ABB RobotStudio station: Lab3.rsstn

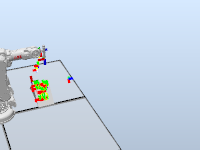
Station Lab1 (saved by RobotStudio 22.1.9826.0)
Controller IRB140_6_81
  mechanical unit ROB_1: IRB140_6_81_C_03, 6 joints, base frame (0, 0, 0) mm
Layout (positions relative to the parent item):
  - IRB140_6_81_C_03 [mechanism, from Robots\IRB140_6_81_C_G_03.rslib] at (0, 0, 0) mm; joint values [0.1206, 0.0069, 0.5145, 0.2099, -0.5334, 0.5073] (rad or m)
  - TableroBorrable [part, from Libraries\TableroBorrable.rslib] at (618.49, 141.25, 150.15) mm
  - Portamarcador [mechanism, from Libraries\Portamarcador.rslib] at (515, 0, 712) mm, rotated rx 0 ry 90 rz 0 deg
Attachment: Portamarcador is attached to IRB140_6_81_C_03 / Link6
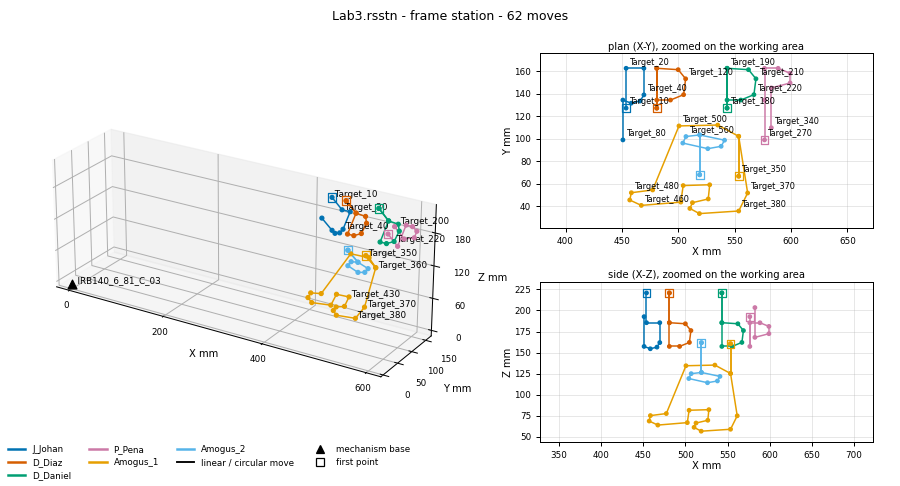
[picture p0: tool path of Lab3.rsstn in frame station, 62 of 66 moves have a stored position in this frame; points joined in program order, loops and branches not executed]
Targets, tools, work objects and paths stored in the station, written as RAPID:
! task T_ROB1
MODULE Module1
  PROC main()
    SetDO SalDO_1,0;
    WaitDI EntDI_1,1;
    SetDO SalDO_1,1;
    Aproximate;
    J_Johan;
    D_Diaz;
    D_Daniel;
    P_Pena;
    Amogus_1;
    Amogus_2;
    GoHome_;
    main;
  ENDPROC
  PROC J_Johan()
    MoveL Target_10,v30,z10,Portamarcador\WObj:=Tablero;
    MoveL Target_20,v30,z10,Portamarcador\WObj:=Tablero;
    MoveL Target_30,v30,z10,Portamarcador\WObj:=Tablero;
    MoveL Target_40,v30,z10,Portamarcador\WObj:=Tablero;
    MoveL Target_50,v30,z10,Portamarcador\WObj:=Tablero;
    MoveL Target_60,v30,z10,Portamarcador\WObj:=Tablero;
    MoveL Target_70,v30,z10,Portamarcador\WObj:=Tablero;
    MoveL Target_80,v30,z10,Portamarcador\WObj:=Tablero;
  ENDPROC
  PROC D_Diaz()
    MoveL Target_90,v30,z10,Portamarcador\WObj:=Tablero;
    MoveL Target_100,v30,z10,Portamarcador\WObj:=Tablero;
    MoveL Target_110,v30,z10,Portamarcador\WObj:=Tablero;
    MoveL Target_120,v30,z10,Portamarcador\WObj:=Tablero;
    MoveL Target_130,v30,z10,Portamarcador\WObj:=Tablero;
    MoveL Target_140,v30,z10,Portamarcador\WObj:=Tablero;
    MoveL Target_150,v30,z10,Portamarcador\WObj:=Tablero;
    MoveL Target_160,v30,z10,Portamarcador\WObj:=Tablero;
    MoveL Target_170,v30,z10,Portamarcador\WObj:=Tablero;
  ENDPROC
  PROC D_Daniel()
    MoveL Target_180,v30,z10,Portamarcador\WObj:=Tablero;
    MoveL Target_190,v30,z10,Portamarcador\WObj:=Tablero;
    MoveL Target_200,v30,z10,Portamarcador\WObj:=Tablero;
    MoveL Target_210,v30,z10,Portamarcador\WObj:=Tablero;
    MoveL Target_220,v30,z10,Portamarcador\WObj:=Tablero;
    MoveL Target_230,v30,z10,Portamarcador\WObj:=Tablero;
    MoveL Target_240,v30,z10,Portamarcador\WObj:=Tablero;
    MoveL Target_250,v30,z10,Portamarcador\WObj:=Tablero;
    MoveL Target_260,v30,z10,Portamarcador\WObj:=Tablero;
  ENDPROC
  PROC P_Pena()
    MoveL Target_270,v30,z10,Portamarcador\WObj:=Tablero;
    MoveL Target_280,v30,z10,Portamarcador\WObj:=Tablero;
    MoveL Target_290,v30,z10,Portamarcador\WObj:=Tablero;
    MoveL Target_300,v30,z10,Portamarcador\WObj:=Tablero;
    MoveL Target_310,v30,z10,Portamarcador\WObj:=Tablero;
    MoveL Target_320,v30,z10,Portamarcador\WObj:=Tablero;
    MoveL Target_330,v30,z10,Portamarcador\WObj:=Tablero;
    MoveL Target_340,v30,z10,Portamarcador\WObj:=Tablero;
  ENDPROC
  PROC Aproximate()
    MoveAbsJ Home,v30,z10,Portamarcador\WObj:=Tablero;
    MoveJ \Conc,MidPoint2,v30,z10,Portamarcador\WObj:=Tablero;
  ENDPROC
  PROC GoHome_()
    MoveAbsJ Home,v30,z10,Portamarcador\WObj:=Tablero;
  ENDPROC
  PROC Amogus_1()
    MoveL Target_350,v30,z10,Portamarcador\WObj:=Tablero;
    MoveL Target_360,v30,z10,Portamarcador\WObj:=Tablero;
    MoveL Target_370,v30,z10,Portamarcador\WObj:=Tablero;
    MoveL Target_380,v30,z10,Portamarcador\WObj:=Tablero;
    MoveL Target_390,v30,z10,Portamarcador\WObj:=Tablero;
    MoveL Target_400,v30,z10,Portamarcador\WObj:=Tablero;
    MoveL Target_410,v30,z10,Portamarcador\WObj:=Tablero;
    MoveL Target_420,v30,z10,Portamarcador\WObj:=Tablero;
    MoveL Target_430,v30,z10,Portamarcador\WObj:=Tablero;
    MoveL Target_440,v30,z10,Portamarcador\WObj:=Tablero;
    MoveL Target_450,v30,z10,Portamarcador\WObj:=Tablero;
    MoveL Target_460,v30,z10,Portamarcador\WObj:=Tablero;
    MoveL Target_470,v30,z10,Portamarcador\WObj:=Tablero;
    MoveL Target_480,v30,z10,Portamarcador\WObj:=Tablero;
    MoveL Target_490,v30,z10,Portamarcador\WObj:=Tablero;
    MoveL Target_500,v30,z10,Portamarcador\WObj:=Tablero;
    MoveL Target_510,v30,z10,Portamarcador\WObj:=Tablero;
    MoveL Target_520,v30,z10,Portamarcador\WObj:=Tablero;
    MoveL Target_530,v30,z10,Portamarcador\WObj:=Tablero;
  ENDPROC
  PROC Amogus_2()
    MoveL Target_540,v30,z10,Portamarcador\WObj:=Tablero;
    MoveL Target_550,v30,z10,Portamarcador\WObj:=Tablero;
    MoveL Target_560,v30,z10,Portamarcador\WObj:=Tablero;
    MoveL Target_570,v30,z10,Portamarcador\WObj:=Tablero;
    MoveL Target_580,v30,z10,Portamarcador\WObj:=Tablero;
    MoveL Target_590,v30,z10,Portamarcador\WObj:=Tablero;
    MoveL Target_600,v30,z10,Portamarcador\WObj:=Tablero;
    MoveL Target_610,v30,z10,Portamarcador\WObj:=Tablero;
    MoveL Target_620,v30,z10,Portamarcador\WObj:=Tablero;
  ENDPROC
  LOCAL PROC Mant()
    MoveAbsJ PosMant,v100,z100,Portamarcador\WObj:=Tablero;
  ENDPROC
ENDMODULE

! task T_ROB1
MODULE CalibData
  PERS tooldata Portamarcador:=[TRUE,[[105.653,-1.591,36.465],[0.707106781,0,0.707106781,0]],[0.25,[0,0,1],[1,0,0,0],0,0,0]];
  TASK PERS wobjdata Tablero:=[FALSE,TRUE,"",[[0,0,0],[1,0,0,0]],[[431.492,204.933,227.769],[0.270598807,-0.653281169,-0.653281169,-0.270598807]]];
ENDMODULE

! task T_ROB1
MODULE GoHome
  CONST jointtarget Home:=[[0,0,0,0,0,0],[9E+09,9E+09,9E+09,9E+09,9E+09,9E+09]];
  CONST robtarget Target_10:=[[-59.887841644,22.215507517,-50.081855147],[0.707106781,0.00000082,-0.00000082,-0.707106781],[0,0,0,1],[9E+09,9E+09,9E+09,9E+09,9E+09,9E+09]];
  CONST robtarget Target_20:=[[-59.887957505,22.215507517,-0.081855147],[0.707106781,0.00000082,-0.00000082,-0.707106781],[0,0,0,1],[9E+09,9E+09,9E+09,9E+09,9E+09,9E+09]];
  CONST robtarget Target_30:=[[-59.887957505,38.001461443,-0.081855147],[0.707106781,0.00000082,-0.00000082,-0.707106781],[0,0,0,1],[9E+09,9E+09,9E+09,9E+09,9E+09,9E+09]];
  CONST robtarget Target_40:=[[-93.271368484,38.001461443,-0.081932504],[0.707106781,0.000000819,-0.000000819,-0.707106781],[0,0,0,1],[9E+09,9E+09,9E+09,9E+09,9E+09,9E+09]];
  CONST robtarget Target_50:=[[-100.93542349,34.650363976,-0.081950263],[0.707106781,0.00000082,-0.000000819,-0.707106781],[0,0,0,1],[9E+09,9E+09,9E+09,9E+09,9E+09,9E+09]];
  CONST robtarget Target_60:=[[-103.679130867,26.748486782,-0.081956621],[0.707106782,0.00000082,-0.000000819,-0.707106781],[0,0,0,1],[9E+09,9E+09,9E+09,9E+09,9E+09,9E+09]];
  CONST robtarget Target_70:=[[-99.741021774,19.368860088,-0.081947494],[0.707106781,0.000000819,-0.00000082,-0.707106781],[0,0,0,1],[9E+09,9E+09,9E+09,9E+09,9E+09,9E+09]];
  CONST robtarget Target_80:=[[-99.740905914,19.368860088,-50.081947495],[0.707106781,0.000000819,-0.00000082,-0.707106781],[0,0,0,1],[9E+09,9E+09,9E+09,9E+09,9E+09,9E+09]];
  CONST robtarget Target_90:=[[-59.88784141,49.388051159,-50.081855147],[0.707106781,0.00000082,-0.00000082,-0.707106781],[0,0,0,1],[9E+09,9E+09,9E+09,9E+09,9E+09,9E+09]];
  CONST robtarget Target_100:=[[-59.887957271,49.388051159,-0.081855147],[0.707106781,0.00000082,-0.00000082,-0.707106781],[0,0,0,1],[9E+09,9E+09,9E+09,9E+09,9E+09,9E+09]];
  CONST robtarget Target_110:=[[-61.656166444,68.408831548,-0.081859245],[0.707106782,0.00000082,-0.000000819,-0.707106781],[0,0,0,1],[9E+09,9E+09,9E+09,9E+09,9E+09,9E+09]];
  CONST robtarget Target_120:=[[-73.086050217,75.007878021,-0.08188573],[0.707106781,0.000000819,-0.000000819,-0.707106781],[0,0,0,1],[9E+09,9E+09,9E+09,9E+09,9E+09,9E+09]];
  CONST robtarget Target_130:=[[-93.012582397,73.204998124,-0.081931904],[0.707106781,0.000000819,-0.000000819,-0.707106781],[0,0,0,1],[9E+09,9E+09,9E+09,9E+09,9E+09,9E+09]];
  CONST robtarget Target_140:=[[-99.741021774,61.550999266,-0.081947494],[0.707106781,0.00000082,-0.00000082,-0.707106781],[0,0,0,1],[9E+09,9E+09,9E+09,9E+09,9E+09,9E+09]];
  CONST robtarget Target_150:=[[-99.741021774,49.388051159,-0.081947494],[0.707106781,0.00000082,-0.00000082,-0.707106781],[0,0,0,1],[9E+09,9E+09,9E+09,9E+09,9E+09,9E+09]];
  CONST robtarget Target_160:=[[-59.887957271,49.388051159,-0.081855147],[0.707106781,0.000000819,-0.000000819,-0.707106781],[0,0,0,1],[9E+09,9E+09,9E+09,9E+09,9E+09,9E+09]];
  CONST robtarget Target_170:=[[-59.88784141,49.388051159,-50.081855147],[0.707106781,0.000000819,-0.000000819,-0.707106781],[0,0,0,1],[9E+09,9E+09,9E+09,9E+09,9E+09,9E+09]];
  CONST robtarget Target_180:=[[-59.88784141,111.75550847,-50.081855147],[0.707106781,0.00000082,-0.00000082,-0.707106781],[0,0,0,1],[9E+09,9E+09,9E+09,9E+09,9E+09,9E+09]];
  CONST robtarget Target_190:=[[-59.887957271,111.75550847,-0.081855147],[0.707106781,0.00000082,-0.00000082,-0.707106781],[0,0,0,1],[9E+09,9E+09,9E+09,9E+09,9E+09,9E+09]];
  CONST robtarget Target_200:=[[-61.656166444,130.776288859,-0.081859245],[0.707106782,0.00000082,-0.000000819,-0.707106781],[0,0,0,1],[9E+09,9E+09,9E+09,9E+09,9E+09,9E+09]];
  CONST robtarget Target_210:=[[-73.086050217,137.375335333,-0.08188573],[0.707106781,0.000000819,-0.000000819,-0.707106781],[0,0,0,1],[9E+09,9E+09,9E+09,9E+09,9E+09,9E+09]];
  CONST robtarget Target_220:=[[-93.012582397,135.572455435,-0.081931904],[0.707106781,0.000000819,-0.000000819,-0.707106781],[0,0,0,1],[9E+09,9E+09,9E+09,9E+09,9E+09,9E+09]];
  CONST robtarget Target_230:=[[-99.741021774,123.918456577,-0.081947494],[0.707106781,0.00000082,-0.00000082,-0.707106781],[0,0,0,1],[9E+09,9E+09,9E+09,9E+09,9E+09,9E+09]];
  CONST robtarget Target_240:=[[-99.741021774,111.75550847,-0.081947494],[0.707106781,0.00000082,-0.00000082,-0.707106781],[0,0,0,1],[9E+09,9E+09,9E+09,9E+09,9E+09,9E+09]];
  CONST robtarget Target_250:=[[-59.887957271,111.75550847,-0.081855147],[0.707106781,0.000000819,-0.000000819,-0.707106781],[0,0,0,1],[9E+09,9E+09,9E+09,9E+09,9E+09,9E+09]];
  CONST robtarget Target_260:=[[-59.88784141,111.75550847,-50.081855147],[0.707106781,0.000000819,-0.000000819,-0.707106781],[0,0,0,1],[9E+09,9E+09,9E+09,9E+09,9E+09,9E+09]];
  CONST robtarget Target_270:=[[-99.740905914,144.97534301,-50.081947495],[0.707106781,0.000000819,-0.000000819,-0.707106781],[0,0,0,1],[9E+09,9E+09,9E+09,9E+09,9E+09,9E+09]];
  CONST robtarget Target_280:=[[-99.741021774,144.97534301,-0.081947494],[0.707106781,0.000000819,-0.000000819,-0.707106781],[0,0,0,1],[9E+09,9E+09,9E+09,9E+09,9E+09,9E+09]];
  CONST robtarget Target_290:=[[-59.983167415,144.97534301,-0.081855368],[0.707106781,0.000000819,-0.000000819,-0.707106781],[0,0,0,1],[9E+09,9E+09,9E+09,9E+09,9E+09,9E+09]];
  CONST robtarget Target_300:=[[-59.983167415,157.043081207,-0.081855368],[0.707106781,0.00000082,-0.00000082,-0.707106781],[0,0,0,1],[9E+09,9E+09,9E+09,9E+09,9E+09,9E+09]];
  CONST robtarget Target_310:=[[-66.114081356,167.662135648,-0.081869575],[0.707106781,0.000000819,-0.000000819,-0.707106781],[0,0,0,1],[9E+09,9E+09,9E+09,9E+09,9E+09,9E+09]];
  CONST robtarget Target_320:=[[-78.375909236,167.662135648,-0.081897988],[0.707106781,0.000000819,-0.000000819,-0.707106781],[0,0,0,1],[9E+09,9E+09,9E+09,9E+09,9E+09,9E+09]];
  CONST robtarget Target_330:=[[-84.506823176,151.009212109,-0.081912194],[0.707106781,0.00000082,-0.00000082,-0.707106781],[0,0,0,1],[9E+09,9E+09,9E+09,9E+09,9E+09,9E+09]];
  CONST robtarget Target_340:=[[-84.506707316,151.009212109,-50.081912194],[0.707106781,0.00000082,-0.00000082,-0.707106781],[0,0,0,1],[9E+09,9E+09,9E+09,9E+09,9E+09,9E+09]];
  CONST robtarget Target_350:=[[-145.225874554,122.068654602,-50.082052893],[0.707106781,0.000000819,-0.000000819,-0.707106781],[-1,-1,0,1],[9E+09,9E+09,9E+09,9E+09,9E+09,9E+09]];
  CONST robtarget Target_360:=[[-145.225990414,122.068654602,-0.082052893],[0.707106781,0.000000819,-0.000000819,-0.707106781],[0,0,0,1],[9E+09,9E+09,9E+09,9E+09,9E+09,9E+09]];
  CONST robtarget Target_370:=[[-216.314272977,130.011265242,-0.08221762],[0.707106782,0.00000082,-0.000000819,-0.707106781],[-1,-1,0,1],[9E+09,9E+09,9E+09,9E+09,9E+09,9E+09]];
  CONST robtarget Target_380:=[[-238.920712,122.070831135,-0.082270004],[0.707106781,0.00000082,-0.00000082,-0.707106781],[-1,-1,0,1],[9E+09,9E+09,9E+09,9E+09,9E+09,9E+09]];
  CONST robtarget Target_390:=[[-242.176963668,87.21495429,-0.082277549],[0.707106781,0.000000819,-0.000000819,-0.707106781],[-1,-1,0,1],[9E+09,9E+09,9E+09,9E+09,9E+09,9E+09]];
  CONST robtarget Target_400:=[[-235.683786475,78.752058887,-0.082262503],[0.707106781,0.000000819,-0.000000819,-0.707106781],[-1,-1,0,1],[9E+09,9E+09,9E+09,9E+09,9E+09,9E+09]];
  CONST robtarget Target_410:=[[-228.457991082,81.055519424,-0.082245759],[0.707106781,0.000000819,-0.000000819,-0.707106781],[-1,-1,0,1],[9E+09,9E+09,9E+09,9E+09,9E+09,9E+09]];
  CONST robtarget Target_420:=[[-223.813275477,95.060731266,-0.082234996],[0.707106781,0.000000819,-0.000000819,-0.707106781],[-1,-1,0,1],[9E+09,9E+09,9E+09,9E+09,9E+09,9E+09]];
  CONST robtarget Target_430:=[[-205.993838978,96.347520237,-0.082193705],[0.707106781,0.000000819,-0.00000082,-0.707106782],[-1,-1,0,1],[9E+09,9E+09,9E+09,9E+09,9E+09,9E+09]];
  CONST robtarget Target_440:=[[-207.00309405,72.842237427,-0.082196044],[0.707106782,0.000000819,-0.000000818,-0.707106781],[-1,-1,0,1],[9E+09,9E+09,9E+09,9E+09,9E+09,9E+09]];
  CONST robtarget Target_450:=[[-227.772910705,70.716966245,-0.082244172],[0.707106781,0.000000819,-0.000000819,-0.707106781],[-1,-1,0,1],[9E+09,9E+09,9E+09,9E+09,9E+09,9E+09]];
  CONST robtarget Target_460:=[[-231.882732587,35.693817055,-0.082253695],[0.707106781,0.000000819,-0.000000819,-0.707106781],[-1,-1,0,1],[9E+09,9E+09,9E+09,9E+09,9E+09,9E+09]];
  CONST robtarget Target_470:=[[-225.128328942,25.434710387,-0.082238044],[0.707106781,0.000000819,-0.000000819,-0.707106781],[-1,-1,0,1],[9E+09,9E+09,9E+09,9E+09,9E+09,9E+09]];
  CONST robtarget Target_480:=[[-215.976129925,26.869358271,-0.082216836],[0.707106781,0.00000082,-0.00000082,-0.707106781],[-1,-1,0,1],[9E+09,9E+09,9E+09,9E+09,9E+09,9E+09]];
  CONST robtarget Target_490:=[[-212.521294514,45.774375392,-0.08220883],[0.707106781,0.000000819,-0.000000819,-0.707106781],[-1,-1,0,1],[9E+09,9E+09,9E+09,9E+09,9E+09,9E+09]];
  CONST robtarget Target_500:=[[-132.204623558,69.10534384,-0.08202272],[0.707106781,0.000000819,-0.00000082,-0.707106782],[0,0,0,1],[9E+09,9E+09,9E+09,9E+09,9E+09,9E+09]];
  CONST robtarget Target_510:=[[-131.099190925,103.471454414,-0.082020159],[0.707106781,0.000000819,-0.000000819,-0.707106781],[0,0,0,1],[9E+09,9E+09,9E+09,9E+09,9E+09,9E+09]];
  CONST robtarget Target_520:=[[-145.225990414,122.068654602,-0.082052893],[0.707106781,0.000000819,-0.000000819,-0.707106781],[0,0,0,1],[9E+09,9E+09,9E+09,9E+09,9E+09,9E+09]];
  CONST robtarget Target_530:=[[-145.225874554,122.068654602,-50.082052893],[0.707106781,0.000000819,-0.000000819,-0.707106781],[-1,-1,0,1],[9E+09,9E+09,9E+09,9E+09,9E+09,9E+09]];
  CONST robtarget Target_540:=[[-143.491221184,87.474940519,-50.082048873],[0.707106781,0.000000819,-0.000000819,-0.707106781],[-1,-1,0,1],[9E+09,9E+09,9E+09,9E+09,9E+09,9E+09]];
  CONST robtarget Target_550:=[[-143.491337044,87.474940519,-0.082048874],[0.707106781,0.000000819,-0.000000819,-0.707106781],[0,0,0,1],[9E+09,9E+09,9E+09,9E+09,9E+09,9E+09]];
  CONST robtarget Target_560:=[[-145.497156615,75.291484437,-0.082053521],[0.707106781,0.000000819,-0.000000819,-0.707106781],[0,0,0,1],[9E+09,9E+09,9E+09,9E+09,9E+09,9E+09]];
  CONST robtarget Target_570:=[[-153.701887033,72.48506132,-0.082072534],[0.707106781,0.000000819,-0.00000082,-0.707106782],[0,0,0,1],[9E+09,9E+09,9E+09,9E+09,9E+09,9E+09]];
  CONST robtarget Target_580:=[[-160.745274412,94.690565784,-0.082088855],[0.707106782,0.00000082,-0.000000819,-0.707106781],[0,0,0,1],[9E+09,9E+09,9E+09,9E+09,9E+09,9E+09]];
  CONST robtarget Target_590:=[[-157.752837767,106.504530415,-0.082081921],[0.707106782,0.000000819,-0.000000818,-0.707106781],[0,0,0,1],[9E+09,9E+09,9E+09,9E+09,9E+09,9E+09]];
  CONST robtarget Target_600:=[[-150.089305159,109.52469583,-0.082064163],[0.707106781,0.000000819,-0.000000819,-0.707106781],[0,0,0,1],[9E+09,9E+09,9E+09,9E+09,9E+09,9E+09]];
  CONST robtarget Target_610:=[[-143.491337044,87.474940519,-0.082048874],[0.707106781,0.000000819,-0.000000819,-0.707106781],[0,0,0,1],[9E+09,9E+09,9E+09,9E+09,9E+09,9E+09]];
  CONST robtarget Target_620:=[[-143.491221184,87.474940519,-50.082048873],[0.707106781,0.000000819,-0.000000819,-0.707106781],[-1,-1,0,1],[9E+09,9E+09,9E+09,9E+09,9E+09,9E+09]];
  CONST jointtarget PosMant:=[[-28,50,-40,0,-20,0],[9E+09,9E+09,9E+09,9E+09,9E+09,9E+09]];
ENDMODULE

